TYPE U_MOVER_STATE :
UNION
  stState             : ARRAY[1..MAX_MOVER] OF ST_MOVER_STATE;

  byState   AT %I*    : ARRAY[1..MAX_MOVER] OF
                        ARRAY[1..SIZEOF(ST_MOVER_STATE)] OF BYTE;
END_UNION
END_TYPE

(* stored: Version 1.1.0.1
   DUT U_MOVER_STATE: Id {837b86ab-15f7-4001-961e-1cf764078fa2} *)
